PROGRAM PRG_4_LOG
VAR
    fbLogHandler: FB_LogHandler;
END_VAR

fbLogHandler();

END_PROGRAM

(* stored: Version 1.1.0.1, ProductVersion 3.1.4022.18
   POU PRG_4_LOG: Id {e421df47-5cc5-4e2e-af84-df201b3be92d}, SpecialFunc None *)
